LIN {X 0,Y 183.418,Z 1201.036,A -85,B 0,C 180,E1 27269.998,E2 27269.998} C_VEL
LIN {X 0,Y 183.226,Z 1199.826,A -85,B 0,C 180,E1 27279.492,E2 27279.492} C_VEL
LIN {X 0,Y 186.448,Z 1195.295,A -85,B 0,C 180,E1 27291.681,E2 27291.681} C_VEL
LIN {X 0,Y 197.947,Z 1184.674,A -85,B 0,C 180,E1 27306.27,E2 27306.27} C_VEL
LIN {X 0,Y 217.326,Z 1169.341,A -85,B 0,C 180,E1 27318.341,E2 27318.341} C_VEL
LIN {X 0,Y 246.49,Z 1146.185,A -85,B 0,C 180,E1 27329.12,E2 27329.12} C_VEL
LIN {X 0,Y 277.502,Z 1119.353,A -85,B 0,C 180,E1 27336.61,E2 27336.61} C_VEL
LIN {X 0,Y 311.114,Z 1086.295,A -85,B 0,C 180,E1 27342.398,E2 27342.398} C_VEL
LIN {X 0,Y 342.028,Z 1050.422,A -85,B 0,C 180,E1 27346.399,E2 27346.399} C_VEL
LIN {X 0,Y 359.417,Z 1027.318,A -85,B 0,C 180,E1 27348.285,E2 27348.285} C_VEL
LIN {X 0,Y 360.437,Z 1023.489,A -85,B 0,C 180,E1 27349.768,E2 27349.768} C_VEL
LIN {X 0,Y 361.093,Z 1015.57,A -85,B 0,C 180,E1 27355.186,E2 27355.186} C_VEL
LIN {X 0,Y 361.858,Z 1011.871,A -85,B 0,C 180,E1 27359.986,E2 27359.986} C_VEL
LIN {X 0,Y 359.734,Z 1016.107,A -85,B 0,C 180,E1 27365.978,E2 27365.978} C_VEL
LIN {X 0,Y 357.801,Z 1024.145,A -85,B 0,C 180,E1 27371.424,E2 27371.424} C_VEL
LIN {X 0,Y 356.491,Z 1027.72,A -85,B 0,C 180,E1 27372.861,E2 27372.861} C_VEL
LIN {X 0,Y 326.897,Z 1064.503,A -85,B 0,C 180,E1 27376.431,E2 27376.431} C_VEL
LIN {X 0,Y 295.294,Z 1097.247,A -85,B 0,C 180,E1 27381.232,E2 27381.232} C_VEL
LIN {X 0,Y 262.763,Z 1126.328,A -85,B 0,C 180,E1 27387.865,E2 27387.865} C_VEL
LIN {X 0,Y 231.737,Z 1150.541,A -85,B 0,C 180,E1 27397.047,E2 27397.047} C_VEL
LIN {X 0,Y 223.281,Z 1156.799,A -85,B 0,C 180,E1 27400.412,E2 27400.412} C_VEL
LIN {X 0,Y 211.981,Z 1163.134,A -85,B 0,C 180,E1 27403.536,E2 27403.536} C_VEL
LIN {X 0,Y 201.181,Z 1168.751,A -85,B 0,C 180,E1 27407.047,E2 27407.047} C_VEL
LIN {X 0,Y 184.669,Z 1180.419,A -85,B 0,C 180,E1 27420.598,E2 27420.598} C_VEL
LIN {X 0,Y 176.715,Z 1187.063,A -85,B 0,C 180,E1 27435.138,E2 27435.138} C_VEL
LIN {X 0,Y 175.238,Z 1188.956,A -85,B 0,C 180,E1 27445.056,E2 27445.056} C_VEL
LIN {X 0,Y 175.45,Z 1189.257,A -85,B 0,C 180,E1 27450.002,E2 27450.002} C_VEL
LIN {X 0,Y 175.659,Z 1188.194,A -85,B 0,C 180,E1 27459.91,E2 27459.91} C_VEL
LIN {X 0,Y 179.978,Z 1184.048,A -85,B 0,C 180,E1 27472.636,E2 27472.636} C_VEL
LIN {X 0,Y 191.782,Z 1175.244,A -85,B 0,C 180,E1 27486.227,E2 27486.227} C_VEL
LIN {X 0,Y 211.897,Z 1161.357,A -85,B 0,C 180,E1 27498.489,E2 27498.489} C_VEL
LIN {X 0,Y 239.263,Z 1141.674,A -85,B 0,C 180,E1 27508.501,E2 27508.501} C_VEL
LIN {X 0,Y 271.981,Z 1115.727,A -85,B 0,C 180,E1 27516.456,E2 27516.456} C_VEL
LIN {X 0,Y 305.801,Z 1084.371,A -85,B 0,C 180,E1 27522.269,E2 27522.269} C_VEL
LIN {X 0,Y 337.194,Z 1050.092,A -85,B 0,C 180,E1 27526.393,E2 27526.393} C_VEL
LIN {X 0,Y 351.788,Z 1031.697,A -85,B 0,C 180,E1 27528.002,E2 27528.002} C_VEL
LIN {X 0,Y 353.629,Z 1025.8,A -85,B 0,C 180,E1 27531.206,E2 27531.206} C_VEL
LIN {X 0,Y 355.183,Z 1021.103,A -85,B 0,C 180,E1 27535.134,E2 27535.134} C_VEL
LIN {X 0,Y 356.99,Z 1017.989,A -85,B 0,C 180,E1 27540.014,E2 27540.014} C_VEL
LIN {X 0,Y 356.017,Z 1023.243,A -85,B 0,C 180,E1 27546.105,E2 27546.105} C_VEL
LIN {X 0,Y 355.109,Z 1030.41,A -85,B 0,C 180,E1 27550.677,E2 27550.677} C_VEL
LIN {X 0,Y 325.133,Z 1067.904,A -85,B 0,C 180,E1 27554.017,E2 27554.017} C_VEL
LIN {X 0,Y 292.851,Z 1101.689,A -85,B 0,C 180,E1 27558.503,E2 27558.503} C_VEL
LIN {X 0,Y 258.573,Z 1132.56,A -85,B 0,C 180,E1 27565.062,E2 27565.062} C_VEL
LIN {X 0,Y 228.636,Z 1156.349,A -85,B 0,C 180,E1 27573.342,E2 27573.342} C_VEL
LIN {X 0,Y 201.93,Z 1176.328,A -85,B 0,C 180,E1 27585.022,E2 27585.022} C_VEL
LIN {X 0,Y 184.29,Z 1189.982,A -85,B 0,C 180,E1 27599.056,E2 27599.056} C_VEL
LIN {X 0,Y 177.725,Z 1196.4,A -85,B 0,C 180,E1 27610.114,E2 27610.114} C_VEL
LIN {X 0,Y 175.342,Z 1199.552,A -85,B 0,C 180,E1 27620.072,E2 27620.072} C_VEL
LIN {X 0,Y 175.506,Z 1200.777,A -85,B 0,C 180,E1 27629.998,E2 27629.998} C_VEL
LIN {X 0,Y 175.34,Z 1199.564,A -85,B 0,C 180,E1 27639.923,E2 27639.923} C_VEL
LIN {X 0,Y 178.183,Z 1195.845,A -85,B 0,C 180,E1 27651.053,E2 27651.053} C_VEL
LIN {X 0,Y 189.458,Z 1185.834,A -85,B 0,C 180,E1 27666.125,E2 27666.125} C_VEL
LIN {X 0,Y 210.379,Z 1170.234,A -85,B 0,C 180,E1 27679.33,E2 27679.33} C_VEL
LIN {X 0,Y 240.858,Z 1147.022,A -85,B 0,C 180,E1 27690.408,E2 27690.408} C_VEL
LIN {X 0,Y 271.953,Z 1121.223,A -85,B 0,C 180,E1 27697.745,E2 27697.745} C_VEL
LIN {X 0,Y 307.104,Z 1087.646,A -85,B 0,C 180,E1 27703.633,E2 27703.633} C_VEL
LIN {X 0,Y 339.058,Z 1051.582,A -85,B 0,C 180,E1 27707.614,E2 27707.614} C_VEL
LIN {X 0,Y 355.138,Z 1030.656,A -85,B 0,C 180,E1 27709.326,E2 27709.326} C_VEL
LIN {X 0,Y 356.13,Z 1023.435,A -85,B 0,C 180,E1 27713.897,E2 27713.897} C_VEL
LIN {X 0,Y 357.106,Z 1018.216,A -85,B 0,C 180,E1 27719.986,E2 27719.986} C_VEL
LIN {X 0,Y 354.832,Z 1022.647,A -85,B 0,C 180,E1 27726.097,E2 27726.097} C_VEL
LIN {X 0,Y 352.474,Z 1030.744,A -85,B 0,C 180,E1 27731.588,E2 27731.588} C_VEL
LIN {X 0,Y 349.194,Z 1035.472,A -85,B 0,C 180,E1 27732.186,E2 27732.186} C_VEL
LIN {X 0,Y 318.089,Z 1071.841,A -85,B 0,C 180,E1 27735.916,E2 27735.916} C_VEL
LIN {X 0,Y 285.251,Z 1104.275,A -85,B 0,C 180,E1 27740.988,E2 27740.988} C_VEL
LIN {X 0,Y 252.697,Z 1131.538,A -85,B 0,C 180,E1 27747.813,E2 27747.813} C_VEL
LIN {X 0,Y 223.071,Z 1153.62,A -85,B 0,C 180,E1 27756.775,E2 27756.775} C_VEL
LIN {X 0,Y 201.181,Z 1168.751,A -85,B 0,C 180,E1 27767.047,E2 27767.047} C_VEL
LIN {X 0,Y 190.976,Z 1173.788,A -85,B 0,C 180,E1 27770.964,E2 27770.964} C_VEL
LIN {X 0,Y 181.496,Z 1178.028,A -85,B 0,C 180,E1 27775.315,E2 27775.315} C_VEL
LIN {X 0,Y 170.975,Z 1185.702,A -85,B 0,C 180,E1 27789.299,E2 27789.299} C_VEL
LIN {X 0,Y 167.334,Z 1189.216,A -85,B 0,C 180,E1 27804.821,E2 27804.821} C_VEL
LIN {X 0,Y 167.543,Z 1189.516,A -85,B 0,C 180,E1 27810.003,E2 27810.003} C_VEL
LIN {X 0,Y 167.837,Z 1188.455,A -85,B 0,C 180,E1 27820.376,E2 27820.376} C_VEL
LIN {X 0,Y 173.857,Z 1183.357,A -85,B 0,C 180,E1 27835.762,E2 27835.762} C_VEL
LIN {X 0,Y 188.248,Z 1173.634,A -85,B 0,C 180,E1 27849.957,E2 27849.957} C_VEL
LIN {X 0,Y 212.732,Z 1157.426,A -85,B 0,C 180,E1 27862.766,E2 27862.766} C_VEL
LIN {X 0,Y 243.562,Z 1135.829,A -85,B 0,C 180,E1 27872.461,E2 27872.461} C_VEL
LIN {X 0,Y 277.925,Z 1108.195,A -85,B 0,C 180,E1 27879.707,E2 27879.707} C_VEL
LIN {X 0,Y 309.381,Z 1078.804,A -85,B 0,C 180,E1 27884.549,E2 27884.549} C_VEL
LIN {X 0,Y 341.478,Z 1042.944,A -85,B 0,C 180,E1 27888.385,E2 27888.385} C_VEL
LIN {X 0,Y 347.471,Z 1035.414,A -85,B 0,C 180,E1 27889.151,E2 27889.151} C_VEL
LIN {X 0,Y 350.105,Z 1027.407,A -85,B 0,C 180,E1 27895.063,E2 27895.063} C_VEL
LIN {X 0,Y 352.178,Z 1024.309,A -85,B 0,C 180,E1 27900.014,E2 27900.014} C_VEL
LIN {X 0,Y 350.951,Z 1029.552,A -85,B 0,C 180,E1 27906.193,E2 27906.193} C_VEL
LIN {X 0,Y 350.216,Z 1034.617,A -85,B 0,C 180,E1 27909.607,E2 27909.607} C_VEL
LIN {X 0,Y 319.882,Z 1071.453,A -85,B 0,C 180,E1 27913.008,E2 27913.008} C_VEL
LIN {X 0,Y 285.546,Z 1105.885,A -85,B 0,C 180,E1 27917.714,E2 27917.714} C_VEL
LIN {X 0,Y 252.287,Z 1134.637,A -85,B 0,C 180,E1 27924.013,E2 27924.013} C_VEL
LIN {X 0,Y 220.335,Z 1158.844,A -85,B 0,C 180,E1 27932.842,E2 27932.842} C_VEL
LIN {X 0,Y 193.955,Z 1177.619,A -85,B 0,C 180,E1 27944.552,E2 27944.552} C_VEL
LIN {X 0,Y 176.012,Z 1190.711,A -85,B 0,C 180,E1 27959.195,E2 27959.195} C_VEL
LIN {X 0,Y 170.118,Z 1196.133,A -85,B 0,C 180,E1 27969.185,E2 27969.185} C_VEL
LIN {X 0,Y 167.202,Z 1200.084,A -85,B 0,C 180,E1 27984.009,E2 27984.009} C_VEL
LIN {X 0,Y 167.594,Z 1200.517,A -85,B 0,C 180,E1 27989.997,E2 27989.997} C_VEL
LIN {X 0,Y 167.484,Z 1199.302,A -85,B 0,C 180,E1 28000.393,E2 28000.393} C_VEL
LIN {X 0,Y 171.231,Z 1194.909,A -85,B 0,C 180,E1 28013.396,E2 28013.396} C_VEL
LIN {X 0,Y 184.708,Z 1184.247,A -85,B 0,C 180,E1 28029.173,E2 28029.173} C_VEL
LIN {X 0,Y 206.114,Z 1169.15,A -85,B 0,C 180,E1 28041.594,E2 28041.594} C_VEL
LIN {X 0,Y 238.305,Z 1145.637,A -85,B 0,C 180,E1 28052.588,E2 28052.588} C_VEL
LIN {X 0,Y 271.532,Z 1118.598,A -85,B 0,C 180,E1 28059.899,E2 28059.899} C_VEL
LIN {X 0,Y 306.256,Z 1086.014,A -85,B 0,C 180,E1 28065.312,E2 28065.312} C_VEL
LIN {X 0,Y 338.54,Z 1049.89,A -85,B 0,C 180,E1 28069.104,E2 28069.104} C_VEL
LIN {X 0,Y 350.233,Z 1034.886,A -85,B 0,C 180,E1 28070.393,E2 28070.393} C_VEL
LIN {X 0,Y 351.273,Z 1028.329,A -85,B 0,C 180,E1 28075.051,E2 28075.051} C_VEL
LIN {X 0,Y 352.285,Z 1024.526,A -85,B 0,C 180,E1 28079.986,E2 28079.986} C_VEL
LIN {X 0,Y 349.637,Z 1029.052,A -85,B 0,C 180,E1 28086.266,E2 28086.266} C_VEL
LIN {X 0,Y 347.681,Z 1035.385,A -85,B 0,C 180,E1 28090.695,E2 28090.695} C_VEL
LIN {X 0,Y 339.539,Z 1045.579,A -85,B 0,C 180,E1 28091.739,E2 28091.739} C_VEL
LIN {X 0,Y 308.214,Z 1080.186,A -85,B 0,C 180,E1 28095.511,E2 28095.511} C_VEL
LIN {X 0,Y 273.406,Z 1112.194,A -85,B 0,C 180,E1 28101.002,E2 28101.002} C_VEL
LIN {X 0,Y 240.246,Z 1138.343,A -85,B 0,C 180,E1 28108.292,E2 28108.292} C_VEL
LIN {X 0,Y 208.56,Z 1160.321,A -85,B 0,C 180,E1 28118.845,E2 28118.845} C_VEL
LIN {X 0,Y 185.105,Z 1175.622,A -85,B 0,C 180,E1 28132.249,E2 28132.249} C_VEL
LIN {X 0,Y 181.496,Z 1178.028,A -85,B 0,C 180,E1 28135.315,E2 28135.315} C_VEL
LIN {X 0,Y 172.831,Z 1181.712,A -85,B 0,C 180,E1 28140.101,E2 28140.101} C_VEL
LIN {X 0,Y 165.053,Z 1184.714,A -85,B 0,C 180,E1 28145.359,E2 28145.359} C_VEL
LIN {X 0,Y 159.959,Z 1188.748,A -85,B 0,C 180,E1 28159.112,E2 28159.112} C_VEL
LIN {X 0,Y 159.653,Z 1189.775,A -85,B 0,C 180,E1 28170.003,E2 28170.003} C_VEL
LIN {X 0,Y 159.995,Z 1188.718,A -85,B 0,C 180,E1 28180.891,E2 28180.891} C_VEL
LIN {X 0,Y 166.618,Z 1183.622,A -85,B 0,C 180,E1 28196.969,E2 28196.969} C_VEL
LIN {X 0,Y 182.326,Z 1173.712,A -85,B 0,C 180,E1 28211.811,E2 28211.811} C_VEL
LIN {X 0,Y 208.771,Z 1157.113,A -85,B 0,C 180,E1 28224.926,E2 28224.926} C_VEL
LIN {X 0,Y 239.408,Z 1136.456,A -85,B 0,C 180,E1 28234.085,E2 28234.085} C_VEL
LIN {X 0,Y 275.19,Z 1108.466,A -85,B 0,C 180,E1 28241.308,E2 28241.308} C_VEL
LIN {X 0,Y 307.049,Z 1079.349,A -85,B 0,C 180,E1 28245.977,E2 28245.977} C_VEL
LIN {X 0,Y 339.271,Z 1044.02,A -85,B 0,C 180,E1 28249.649,E2 28249.649} C_VEL
LIN {X 0,Y 342.654,Z 1039.794,A -85,B 0,C 180,E1 28250.177,E2 28250.177} C_VEL
LIN {X 0,Y 344.976,Z 1033.672,A -85,B 0,C 180,E1 28254.989,E2 28254.989} C_VEL
LIN {X 0,Y 347.141,Z 1030.439,A -85,B 0,C 180,E1 28260.014,E2 28260.014} C_VEL
LIN {X 0,Y 345.802,Z 1035.856,A -85,B 0,C 180,E1 28266.286,E2 28266.286} C_VEL
LIN {X 0,Y 345.346,Z 1038.832,A -85,B 0,C 180,E1 28268.419,E2 28268.419} C_VEL
LIN {X 0,Y 342.797,Z 1042.436,A -85,B 0,C 180,E1 28268.971,E2 28268.971} C_VEL
LIN {X 0,Y 309.616,Z 1080.038,A -85,B 0,C 180,E1 28272.54,E2 28272.54} C_VEL
LIN {X 0,Y 276.824,Z 1111.353,A -85,B 0,C 180,E1 28277.114,E2 28277.114} C_VEL
LIN {X 0,Y 240.003,Z 1141.226,A -85,B 0,C 180,E1 28284.302,E2 28284.302} C_VEL
LIN {X 0,Y 208.261,Z 1163.884,A -85,B 0,C 180,E1 28293.675,E2 28293.675} C_VEL
LIN {X 0,Y 181.804,Z 1181.601,A -85,B 0,C 180,E1 28306.704,E2 28306.704} C_VEL
LIN {X 0,Y 166.925,Z 1192.112,A -85,B 0,C 180,E1 28320.422,E2 28320.422} C_VEL
LIN {X 0,Y 160.615,Z 1197.691,A -85,B 0,C 180,E1 28333.603,E2 28333.603} C_VEL
LIN {X 0,Y 159.344,Z 1199.885,A -85,B 0,C 180,E1 28344.556,E2 28344.556} C_VEL
LIN {X 0,Y 159.704,Z 1200.258,A -85,B 0,C 180,E1 28349.997,E2 28349.997} C_VEL
LIN {X 0,Y 159.61,Z 1199.039,A -85,B 0,C 180,E1 28360.912,E2 28360.912} C_VEL
LIN {X 0,Y 163.791,Z 1194.642,A -85,B 0,C 180,E1 28374.527,E2 28374.527} C_VEL
LIN {X 0,Y 178.314,Z 1184.017,A -85,B 0,C 180,E1 28390.801,E2 28390.801} C_VEL
LIN {X 0,Y 201.123,Z 1168.817,A -85,B 0,C 180,E1 28403.493,E2 28403.493} C_VEL
LIN {X 0,Y 234.583,Z 1145.365,A -85,B 0,C 180,E1 28414.396,E2 28414.396} C_VEL
LIN {X 0,Y 268.796,Z 1118.328,A -85,B 0,C 180,E1 28421.558,E2 28421.558} C_VEL
LIN {X 0,Y 305.061,Z 1084.991,A -85,B 0,C 180,E1 28426.906,E2 28426.906} C_VEL
LIN {X 0,Y 338.823,Z 1047.512,A -85,B 0,C 180,E1 28430.647,E2 28430.647} C_VEL
LIN {X 0,Y 345.344,Z 1039.407,A -85,B 0,C 180,E1 28431.366,E2 28431.366} C_VEL
LIN {X 0,Y 346.403,Z 1033.254,A -85,B 0,C 180,E1 28436.34,E2 28436.34} C_VEL
LIN {X 0,Y 347.248,Z 1030.655,A -85,B 0,C 180,E1 28439.986,E2 28439.986} C_VEL
LIN {X 0,Y 344.48,Z 1035.364,A -85,B 0,C 180,E1 28446.36,E2 28446.36} C_VEL
LIN {X 0,Y 342.916,Z 1039.568,A -85,B 0,C 180,E1 28449.496,E2 28449.496} C_VEL
LIN {X 0,Y 341.986,Z 1041.044,A -85,B 0,C 180,E1 28449.984,E2 28449.984} C_VEL
LIN {X 0,Y 308.561,Z 1077.993,A -85,B 0,C 180,E1 28453.732,E2 28453.732} C_VEL
LIN {X 0,Y 275.072,Z 1108.73,A -85,B 0,C 180,E1 28458.63,E2 28458.63} C_VEL
LIN {X 0,Y 239.268,Z 1136.669,A -85,B 0,C 180,E1 28465.851,E2 28465.851} C_VEL
LIN {X 0,Y 206.737,Z 1158.483,A -85,B 0,C 180,E1 28475.75,E2 28475.75} C_VEL
LIN {X 0,Y 181.917,Z 1174.027,A -85,B 0,C 180,E1 28488.357,E2 28488.357} C_VEL
LIN {X 0,Y 166.587,Z 1183.689,A -85,B 0,C 180,E1 28503.031,E2 28503.031} C_VEL
LIN {X 0,Y 165.053,Z 1184.714,A -85,B 0,C 180,E1 28505.359,E2 28505.359} C_VEL
LIN {X 0,Y 160.242,Z 1186.573,A -85,B 0,C 180,E1 28509.619,E2 28509.619} C_VEL
LIN {X 0,Y 152.607,Z 1188.636,A -85,B 0,C 180,E1 28516.32,E2 28516.32} C_VEL
LIN {X 0,Y 152.35,Z 1188.726,A -85,B 0,C 180,E1 28517.141,E2 28517.141} C_VEL
LIN {X 0,Y 151.743,Z 1190.035,A -85,B 0,C 180,E1 28530.003,E2 28530.003} C_VEL
LIN {X 0,Y 152.168,Z 1188.98,A -85,B 0,C 180,E1 28541.459,E2 28541.459} C_VEL
LIN {X 0,Y 156.867,Z 1185.546,A -85,B 0,C 180,E1 28554.346,E2 28554.346} C_VEL
LIN {X 0,Y 172.503,Z 1176.107,A -85,B 0,C 180,E1 28570.973,E2 28570.973} C_VEL
LIN {X 0,Y 196.444,Z 1162.169,A -85,B 0,C 180,E1 28583.875,E2 28583.875} C_VEL
LIN {X 0,Y 230.049,Z 1140.657,A -85,B 0,C 180,E1 28594.508,E2 28594.508} C_VEL
LIN {X 0,Y 263.658,Z 1116.101,A -85,B 0,C 180,E1 28601.467,E2 28601.467} C_VEL
LIN {X 0,Y 299.879,Z 1084.608,A -85,B 0,C 180,E1 28606.805,E2 28606.805} C_VEL
LIN {X 0,Y 332.328,Z 1050.899,A -85,B 0,C 180,E1 28610.458,E2 28610.458} C_VEL
LIN {X 0,Y 336.705,Z 1045.714,A -85,B 0,C 180,E1 28610.884,E2 28610.884} C_VEL
LIN {X 0,Y 338.021,Z 1043.677,A -85,B 0,C 180,E1 28611.615,E2 28611.615} C_VEL
LIN {X 0,Y 340.938,Z 1037.886,A -85,B 0,C 180,E1 28617.475,E2 28617.475} C_VEL
LIN {X 0,Y 342.105,Z 1036.566,A -85,B 0,C 180,E1 28620.015,E2 28620.015} C_VEL
LIN {X 0,Y 340.561,Z 1042.087,A -85,B 0,C 180,E1 28626.383,E2 28626.383} C_VEL
LIN {X 0,Y 340.181,Z 1043.798,A -85,B 0,C 180,E1 28627.672,E2 28627.672} C_VEL
LIN {X 0,Y 305.455,Z 1082.322,A -85,B 0,C 180,E1 28631.328,E2 28631.328} C_VEL
LIN {X 0,Y 271.242,Z 1113.777,A -85,B 0,C 180,E1 28635.963,E2 28635.963} C_VEL
LIN {X 0,Y 236.17,Z 1141.359,A -85,B 0,C 180,E1 28642.596,E2 28642.596} C_VEL
LIN {X 0,Y 204.395,Z 1163.218,A -85,B 0,C 180,E1 28651.512,E2 28651.512} C_VEL
LIN {X 0,Y 175.581,Z 1181.505,A -85,B 0,C 180,E1 28665.023,E2 28665.023} C_VEL
LIN {X 0,Y 158.08,Z 1193.072,A -85,B 0,C 180,E1 28681.445,E2 28681.445} C_VEL
LIN {X 0,Y 152.905,Z 1197.427,A -85,B 0,C 180,E1 28692.751,E2 28692.751} C_VEL
LIN {X 0,Y 151.441,Z 1199.782,A -85,B 0,C 180,E1 28706.634,E2 28706.634} C_VEL
LIN {X 0,Y 151.448,Z 1199.783,A -85,B 0,C 180,E1 28713.413,E2 28713.413} C_VEL
LIN {X 0,Y 152.901,Z 1197.448,A -85,B 0,C 180,E1 28727.244,E2 28727.244} C_VEL
LIN {X 0,Y 162.327,Z 1190.096,A -85,B 0,C 180,E1 28743.952,E2 28743.952} C_VEL
LIN {X 0,Y 183.516,Z 1176.639,A -85,B 0,C 180,E1 28759.608,E2 28759.608} C_VEL
LIN {X 0,Y 214.42,Z 1156.611,A -85,B 0,C 180,E1 28771.751,E2 28771.751} C_VEL
LIN {X 0,Y 249.177,Z 1131.765,A -85,B 0,C 180,E1 28780.16,E2 28780.16} C_VEL
LIN {X 0,Y 286.715,Z 1100.365,A -85,B 0,C 180,E1 28786.319,E2 28786.319} C_VEL
LIN {X 0,Y 320.047,Z 1067.342,A -85,B 0,C 180,E1 28790.263,E2 28790.263} C_VEL
LIN {X 0,Y 340.258,Z 1043.985,A -85,B 0,C 180,E1 28792.33,E2 28792.33} C_VEL
LIN {X 0,Y 341.548,Z 1038.489,A -85,B 0,C 180,E1 28797.45,E2 28797.45} C_VEL
LIN {X 0,Y 342.211,Z 1036.783,A -85,B 0,C 180,E1 28799.985,E2 28799.985} C_VEL
LIN {X 0,Y 339.167,Z 1041.456,A -85,B 0,C 180,E1 28806.379,E2 28806.379} C_VEL
LIN {X 0,Y 337.889,Z 1044.452,A -85,B 0,C 180,E1 28808.734,E2 28808.734} C_VEL
LIN {X 0,Y 326.122,Z 1058.025,A -85,B 0,C 180,E1 28810.102,E2 28810.102} C_VEL
LIN {X 0,Y 292.161,Z 1092.097,A -85,B 0,C 180,E1 28814.127,E2 28814.127} C_VEL
LIN {X 0,Y 256.786,Z 1121.504,A -85,B 0,C 180,E1 28819.691,E2 28819.691} C_VEL
LIN {X 0,Y 221.694,Z 1146.471,A -85,B 0,C 180,E1 28827.616,E2 28827.616} C_VEL
LIN {X 0,Y 191.794,Z 1164.903,A -85,B 0,C 180,E1 28838.016,E2 28838.016} C_VEL
LIN {X 0,Y 169.317,Z 1178.006,A -85,B 0,C 180,E1 28851.341,E2 28851.341} C_VEL
LIN {X 0,Y 156.027,Z 1186.229,A -85,B 0,C 180,E1 28867.21,E2 28867.21} C_VEL
LIN {X 0,Y 152.35,Z 1188.726,A -85,B 0,C 180,E1 28877.141,E2 28877.141} C_VEL
LIN {X 0,Y 149.463,Z 1189.68,A -85,B 0,C 180,E1 28881.973,E2 28881.973} C_VEL
LIN {X 0,Y 143.783,Z 1190.277,A -85,B 0,C 180,E1 28890.351,E2 28890.351} C_VEL
LIN {X 0,Y 144.349,Z 1189.242,A -85,B 0,C 180,E1 28902.088,E2 28902.088} C_VEL
LIN {X 0,Y 150.329,Z 1185.303,A -85,B 0,C 180,E1 28916.897,E2 28916.897} C_VEL
LIN {X 0,Y 168.326,Z 1175.37,A -85,B 0,C 180,E1 28934.146,E2 28934.146} C_VEL
LIN {X 0,Y 195.503,Z 1160.167,A -85,B 0,C 180,E1 28947.28,E2 28947.28} C_VEL
LIN {X 0,Y 229.718,Z 1138.958,A -85,B 0,C 180,E1 28957.068,E2 28957.068} C_VEL
LIN {X 0,Y 265.483,Z 1112.928,A -85,B 0,C 180,E1 28963.829,E2 28963.829} C_VEL
LIN {X 0,Y 302.055,Z 1081.275,A -85,B 0,C 180,E1 28968.785,E2 28968.785} C_VEL
LIN {X 0,Y 331.696,Z 1050.45,A -85,B 0,C 180,E1 28971.894,E2 28971.894} C_VEL
LIN {X 0,Y 332.878,Z 1048.939,A -85,B 0,C 180,E1 28972.189,E2 28972.189} C_VEL
LIN {X 0,Y 335.59,Z 1043.877,A -85,B 0,C 180,E1 28977.434,E2 28977.434} C_VEL
LIN {X 0,Y 336.892,Z 1042.561,A -85,B 0,C 180,E1 28980.015,E2 28980.015} C_VEL
LIN {X 0,Y 335.279,Z 1047.524,A -85,B 0,C 180,E1 28985.966,E2 28985.966} C_VEL
LIN {X 0,Y 334.778,Z 1048.798,A -85,B 0,C 180,E1 28986.758,E2 28986.758} C_VEL
LIN {X 0,Y 301.437,Z 1084.552,A -85,B 0,C 180,E1 28990.081,E2 28990.081} C_VEL
LIN {X 0,Y 265.694,Z 1116.276,A -85,B 0,C 180,E1 28994.786,E2 28994.786} C_VEL
LIN {X 0,Y 230.499,Z 1142.98,A -85,B 0,C 180,E1 29001.267,E2 29001.267} C_VEL
LIN {X 0,Y 196.334,Z 1165.26,A -85,B 0,C 180,E1 29010.774,E2 29010.774} C_VEL
LIN {X 0,Y 168.213,Z 1182.24,A -85,B 0,C 180,E1 29024.052,E2 29024.052} C_VEL
LIN {X 0,Y 150.951,Z 1192.803,A -85,B 0,C 180,E1 29039.962,E2 29039.962} C_VEL
LIN {X 0,Y 145.206,Z 1197.161,A -85,B 0,C 180,E1 29051.805,E2 29051.805} C_VEL
LIN {X 0,Y 143.513,Z 1199.363,A -85,B 0,C 180,E1 29063.953,E2 29063.953} C_VEL
LIN {X 0,Y 143.88,Z 1199.739,A -85,B 0,C 180,E1 29069.997,E2 29069.997} C_VEL
LIN {X 0,Y 143.9,Z 1198.514,A -85,B 0,C 180,E1 29082.121,E2 29082.121} C_VEL
LIN {X 0,Y 149.11,Z 1194.108,A -85,B 0,C 180,E1 29097.129,E2 29097.129} C_VEL
LIN {X 0,Y 165.07,Z 1184.082,A -85,B 0,C 180,E1 29113.789,E2 29113.789} C_VEL
LIN {X 0,Y 190.247,Z 1169.19,A -85,B 0,C 180,E1 29126.943,E2 29126.943} C_VEL
LIN {X 0,Y 224.909,Z 1146.812,A -85,B 0,C 180,E1 29137.488,E2 29137.488} C_VEL
LIN {X 0,Y 260.749,Z 1120.48,A -85,B 0,C 180,E1 29144.458,E2 29144.458} C_VEL
LIN {X 0,Y 298.136,Z 1087.828,A -85,B 0,C 180,E1 29149.554,E2 29149.554} C_VEL
LIN {X 0,Y 331.191,Z 1053.334,A -85,B 0,C 180,E1 29152.91,E2 29152.91} C_VEL
LIN {X 0,Y 334.77,Z 1049.095,A -85,B 0,C 180,E1 29153.231,E2 29153.231} C_VEL
LIN {X 0,Y 336.235,Z 1044.474,A -85,B 0,C 180,E1 29157.41,E2 29157.41} C_VEL
LIN {X 0,Y 336.979,Z 1042.777,A -85,B 0,C 180,E1 29159.985,E2 29159.985} C_VEL
LIN {X 0,Y 333.697,Z 1047.565,A -85,B 0,C 180,E1 29166.483,E2 29166.483} C_VEL
LIN {X 0,Y 332.952,Z 1049.206,A -85,B 0,C 180,E1 29167.809,E2 29167.809} C_VEL
LIN {X 0,Y 299.915,Z 1083.443,A -85,B 0,C 180,E1 29171.366,E2 29171.366} C_VEL
LIN {X 0,Y 262.037,Z 1115.853,A -85,B 0,C 180,E1 29176.62,E2 29176.62} C_VEL
LIN {X 0,Y 226.514,Z 1141.125,A -85,B 0,C 180,E1 29183.568,E2 29183.568} C_VEL
LIN {X 0,Y 192.871,Z 1161.83,A -85,B 0,C 180,E1 29193.596,E2 29193.596} C_VEL
LIN {X 0,Y 165.449,Z 1176.928,A -85,B 0,C 180,E1 29207.739,E2 29207.739} C_VEL
LIN {X 0,Y 150.301,Z 1185.369,A -85,B 0,C 180,E1 29223.104,E2 29223.104} C_VEL
LIN {X 0,Y 144.318,Z 1189.271,A -85,B 0,C 180,E1 29237.915,E2 29237.915} C_VEL
LIN {X 0,Y 143.783,Z 1190.277,A -85,B 0,C 180,E1 29250.351,E2 29250.351} C_VEL
LIN {X 0,Y 141.037,Z 1190.14,A -85,B 0,C 180,E1 29255.503,E2 29255.503} C_VEL
LIN {X 0,Y 136.867,Z 1189.203,A -85,B 0,C 180,E1 29264.429,E2 29264.429} C_VEL
LIN {X 0,Y 145.349,Z 1184.423,A -85,B 0,C 180,E1 29281.324,E2 29281.324} C_VEL
LIN {X 0,Y 164.419,Z 1174.716,A -85,B 0,C 180,E1 29297.332,E2 29297.332} C_VEL
LIN {X 0,Y 195.011,Z 1158.263,A -85,B 0,C 180,E1 29310.667,E2 29310.667} C_VEL
LIN {X 0,Y 229.691,Z 1137.268,A -85,B 0,C 180,E1 29319.64,E2 29319.64} C_VEL
LIN {X 0,Y 267.76,Z 1109.714,A -85,B 0,C 180,E1 29326.212,E2 29326.212} C_VEL
LIN {X 0,Y 302.466,Z 1079.762,A -85,B 0,C 180,E1 29330.516,E2 29330.516} C_VEL
LIN {X 0,Y 327.027,Z 1054.72,A -85,B 0,C 180,E1 29332.968,E2 29332.968} C_VEL
LIN {X 0,Y 328.228,Z 1053.18,A -85,B 0,C 180,E1 29333.635,E2 29333.635} C_VEL
LIN {X 0,Y 331.562,Z 1048.479,A -85,B 0,C 180,E1 29340.015,E2 29340.015} C_VEL
LIN {X 0,Y 329.994,Z 1053.034,A -85,B 0,C 180,E1 29345.598,E2 29345.598} C_VEL
LIN {X 0,Y 296.687,Z 1087.417,A -85,B 0,C 180,E1 29348.891,E2 29348.891} C_VEL
LIN {X 0,Y 258.54,Z 1120.147,A -85,B 0,C 180,E1 29353.797,E2 29353.797} C_VEL
LIN {X 0,Y 221.87,Z 1146.427,A -85,B 0,C 180,E1 29360.526,E2 29360.526} C_VEL
LIN {X 0,Y 187.852,Z 1167.584,A -85,B 0,C 180,E1 29370.142,E2 29370.142} C_VEL
LIN {X 0,Y 160.609,Z 1182.994,A -85,B 0,C 180,E1 29383.18,E2 29383.18} C_VEL
LIN {X 0,Y 141.894,Z 1193.807,A -85,B 0,C 180,E1 29401.361,E2 29401.361} C_VEL
LIN {X 0,Y 136.083,Z 1198.237,A -85,B 0,C 180,E1 29417.165,E2 29417.165} C_VEL
LIN {X 0,Y 135.979,Z 1199.479,A -85,B 0,C 180,E1 29429.997,E2 29429.997} C_VEL
LIN {X 0,Y 136.08,Z 1198.251,A -85,B 0,C 180,E1 29442.829,E2 29442.829} C_VEL
LIN {X 0,Y 141.896,Z 1193.841,A -85,B 0,C 180,E1 29458.631,E2 29458.631} C_VEL
LIN {X 0,Y 160.61,Z 1183.048,A -85,B 0,C 180,E1 29476.812,E2 29476.812} C_VEL
LIN {X 0,Y 187.872,Z 1167.677,A -85,B 0,C 180,E1 29489.839,E2 29489.839} C_VEL
LIN {X 0,Y 224.938,Z 1144.552,A -85,B 0,C 180,E1 29500.131,E2 29500.131} C_VEL
LIN {X 0,Y 261.3,Z 1118.089,A -85,B 0,C 180,E1 29506.607,E2 29506.607} C_VEL
LIN {X 0,Y 299.446,Z 1085.098,A -85,B 0,C 180,E1 29511.389,E2 29511.389} C_VEL
LIN {X 0,Y 330.055,Z 1053.25,A -85,B 0,C 180,E1 29514.403,E2 29514.403} C_VEL
LIN {X 0,Y 331.658,Z 1048.684,A -85,B 0,C 180,E1 29519.985,E2 29519.985} C_VEL
LIN {X 0,Y 328.253,Z 1053.515,A -85,B 0,C 180,E1 29526.467,E2 29526.467} C_VEL
LIN {X 0,Y 325.853,Z 1056.244,A -85,B 0,C 180,E1 29527.08,E2 29527.08} C_VEL
LIN {X 0,Y 290.324,Z 1091.055,A -85,B 0,C 180,E1 29530.765,E2 29530.765} C_VEL
LIN {X 0,Y 255.096,Z 1119.601,A -85,B 0,C 180,E1 29535.613,E2 29535.613} C_VEL
LIN {X 0,Y 216.487,Z 1145.761,A -85,B 0,C 180,E1 29543.225,E2 29543.225} C_VEL
LIN {X 0,Y 185.919,Z 1163.457,A -85,B 0,C 180,E1 29552.446,E2 29552.446} C_VEL
LIN {X 0,Y 156.879,Z 1178.541,A -85,B 0,C 180,E1 29567.607,E2 29567.607} C_VEL
LIN {X 0,Y 141.283,Z 1186.758,A -85,B 0,C 180,E1 29584.674,E2 29584.674} C_VEL
LIN {X 0,Y 135.766,Z 1190.257,A -85,B 0,C 180,E1 29603.613,E2 29603.613} C_VEL
LIN {X 0,Y 135.897,Z 1190.541,A -85,B 0,C 180,E1 29610.325,E2 29610.325} C_VEL
LIN {X 0,Y 136.867,Z 1189.203,A -85,B 0,C 180,E1 29624.429,E2 29624.429} C_VEL
LIN {X 0,Y 136.625,Z 1188.691,A -85,B 0,C 180,E1 29628.088,E2 29628.088} C_VEL
LIN {X 0,Y 135.029,Z 1186.446,A -85,B 0,C 180,E1 29638.296,E2 29638.296} C_VEL
LIN {X 0,Y 135.54,Z 1186.121,A -85,B 0,C 180,E1 29639.195,E2 29639.195} C_VEL
LIN {X 0,Y 154.68,Z 1176.957,A -85,B 0,C 180,E1 29656.906,E2 29656.906} C_VEL
LIN {X 0,Y 184.241,Z 1162.299,A -85,B 0,C 180,E1 29670.556,E2 29670.556} C_VEL
LIN {X 0,Y 222.121,Z 1140.531,A -85,B 0,C 180,E1 29680.605,E2 29680.605} C_VEL
LIN {X 0,Y 258.114,Z 1116,A -85,B 0,C 180,E1 29686.812,E2 29686.812} C_VEL
LIN {X 0,Y 296.06,Z 1084.708,A -85,B 0,C 180,E1 29691.507,E2 29691.507} C_VEL
LIN {X 0,Y 322.01,Z 1059.301,A -85,B 0,C 180,E1 29694.025,E2 29694.025} C_VEL
LIN {X 0,Y 323.18,Z 1057.881,A -85,B 0,C 180,E1 29694.65,E2 29694.65} C_VEL
LIN {X 0,Y 326.214,Z 1054.382,A -85,B 0,C 180,E1 29700.015,E2 29700.015} C_VEL
LIN {X 0,Y 324.751,Z 1057.797,A -85,B 0,C 180,E1 29704.614,E2 29704.614} C_VEL
LIN {X 0,Y 286.33,Z 1095.532,A -85,B 0,C 180,E1 29708.286,E2 29708.286} C_VEL
LIN {X 0,Y 248.372,Z 1126.018,A -85,B 0,C 180,E1 29713.225,E2 29713.225} C_VEL
LIN {X 0,Y 209.818,Z 1152.121,A -85,B 0,C 180,E1 29720.561,E2 29720.561} C_VEL
LIN {X 0,Y 174.396,Z 1172.422,A -85,B 0,C 180,E1 29731.354,E2 29731.354} C_VEL
LIN {X 0,Y 148.278,Z 1186.239,A -85,B 0,C 180,E1 29745.551,E2 29745.551} C_VEL
LIN {X 0,Y 132.881,Z 1194.796,A -85,B 0,C 180,E1 29762.939,E2 29762.939} C_VEL
LIN {X 0,Y 128.263,Z 1197.973,A -85,B 0,C 180,E1 29776.368,E2 29776.368} C_VEL
LIN {X 0,Y 128.059,Z 1199.219,A -85,B 0,C 180,E1 29789.997,E2 29789.997} C_VEL
LIN {X 0,Y 128.259,Z 1197.987,A -85,B 0,C 180,E1 29803.625,E2 29803.625} C_VEL
LIN {X 0,Y 134.773,Z 1193.573,A -85,B 0,C 180,E1 29820.298,E2 29820.298} C_VEL
LIN {X 0,Y 155.043,Z 1182.776,A -85,B 0,C 180,E1 29839.051,E2 29839.051} C_VEL
LIN {X 0,Y 183.83,Z 1167.406,A -85,B 0,C 180,E1 29852.083,E2 29852.083} C_VEL
LIN {X 0,Y 222.248,Z 1144.28,A -85,B 0,C 180,E1 29862.149,E2 29862.149} C_VEL
LIN {X 0,Y 259.516,Z 1117.821,A -85,B 0,C 180,E1 29868.377,E2 29868.377} C_VEL
LIN {X 0,Y 298.626,Z 1084.564,A -85,B 0,C 180,E1 29872.973,E2 29872.973} C_VEL
LIN {X 0,Y 324.802,Z 1058.01,A -85,B 0,C 180,E1 29875.383,E2 29875.383} C_VEL
LIN {X 0,Y 326.303,Z 1054.575,A -85,B 0,C 180,E1 29879.985,E2 29879.985} C_VEL
LIN {X 0,Y 323.066,Z 1058.428,A -85,B 0,C 180,E1 29885.688,E2 29885.688} C_VEL
LIN {X 0,Y 287.161,Z 1092.894,A -85,B 0,C 180,E1 29889.375,E2 29889.375} C_VEL
LIN {X 0,Y 249.563,Z 1122.307,A -85,B 0,C 180,E1 29894.356,E2 29894.356} C_VEL
LIN {X 0,Y 211.367,Z 1147.278,A -85,B 0,C 180,E1 29901.664,E2 29901.664} C_VEL
LIN {X 0,Y 175.115,Z 1167.004,A -85,B 0,C 180,E1 29912.722,E2 29912.722} C_VEL
LIN {X 0,Y 150.945,Z 1178.809,A -85,B 0,C 180,E1 29925.515,E2 29925.515} C_VEL
LIN {X 0,Y 134.015,Z 1187.023,A -85,B 0,C 180,E1 29943.194,E2 29943.194} C_VEL
LIN {X 0,Y 127.872,Z 1190.518,A -85,B 0,C 180,E1 29963.217,E2 29963.217} C_VEL
LIN {X 0,Y 128.057,Z 1190.812,A -85,B 0,C 180,E1 29970.003,E2 29970.003} C_VEL
LIN {X 0,Y 129.003,Z 1189.565,A -85,B 0,C 180,E1 29984.744,E2 29984.744} C_VEL
LIN {X 0,Y 135.54,Z 1186.121,A -85,B 0,C 180,E1 29999.195,E2 29999.195} C_VEL
LIN {X 0,Y 136.939,Z 1184.97,A -85,B 0,C 180,E1 30002.793,E2 30002.793} C_VEL
LIN {X 0,Y 139.942,Z 1181.382,A -85,B 0,C 180,E1 30012.672,E2 30012.672} C_VEL
LIN {X 0,Y 140.862,Z 1180.974,A -85,B 0,C 180,E1 30013.473,E2 30013.473} C_VEL
LIN {X 0,Y 168.284,Z 1168.433,A -85,B 0,C 180,E1 30028.551,E2 30028.551} C_VEL
LIN {X 0,Y 205.461,Z 1149.081,A -85,B 0,C 180,E1 30039.679,E2 30039.679} C_VEL
LIN {X 0,Y 242.669,Z 1125.886,A -85,B 0,C 180,E1 30046.657,E2 30046.657} C_VEL
LIN {X 0,Y 282.462,Z 1095.849,A -85,B 0,C 180,E1 30051.784,E2 30051.784} C_VEL
LIN {X 0,Y 317.865,Z 1063.077,A -85,B 0,C 180,E1 30055.244,E2 30055.244} C_VEL
LIN {X 0,Y 320.607,Z 1060.066,A -85,B 0,C 180,E1 30060.016,E2 30060.016} C_VEL
LIN {X 0,Y 319.552,Z 1062.296,A -85,B 0,C 180,E1 30063.33,E2 30063.33} C_VEL
LIN {X 0,Y 313.827,Z 1068.457,A -85,B 0,C 180,E1 30064.034,E2 30064.034} C_VEL
LIN {X 0,Y 276.311,Z 1102.759,A -85,B 0,C 180,E1 30067.581,E2 30067.581} C_VEL
LIN {X 0,Y 237.781,Z 1132.083,A -85,B 0,C 180,E1 30072.679,E2 30072.679} C_VEL
LIN {X 0,Y 198.674,Z 1156.65,A -85,B 0,C 180,E1 30080.348,E2 30080.348} C_VEL
LIN {X 0,Y 163.45,Z 1175.722,A -85,B 0,C 180,E1 30091.723,E2 30091.723} C_VEL
LIN {X 0,Y 136.211,Z 1188.97,A -85,B 0,C 180,E1 30108.265,E2 30108.265} C_VEL
LIN {X 0,Y 122.4,Z 1196.364,A -85,B 0,C 180,E1 30128.258,E2 30128.258} C_VEL
LIN {X 0,Y 119.792,Z 1198.579,A -85,B 0,C 180,E1 30142.749,E2 30142.749} C_VEL
LIN {X 0,Y 120.151,Z 1198.96,A -85,B 0,C 180,E1 30149.996,E2 30149.996} C_VEL
LIN {X 0,Y 120.463,Z 1197.724,A -85,B 0,C 180,E1 30164.526,E2 30164.526} C_VEL
LIN {X 0,Y 127.78,Z 1193.305,A -85,B 0,C 180,E1 30182.148,E2 30182.148} C_VEL
LIN {X 0,Y 149.726,Z 1182.504,A -85,B 0,C 180,E1 30201.455,E2 30201.455} C_VEL
LIN {X 0,Y 180.078,Z 1167.133,A -85,B 0,C 180,E1 30214.427,E2 30214.427} C_VEL
LIN {X 0,Y 219.847,Z 1144.01,A -85,B 0,C 180,E1 30224.206,E2 30224.206} C_VEL
LIN {X 0,Y 258.469,Z 1117.162,A -85,B 0,C 180,E1 30230.253,E2 30230.253} C_VEL
LIN {X 0,Y 297.212,Z 1084.762,A -85,B 0,C 180,E1 30234.495,E2 30234.495} C_VEL
LIN {X 0,Y 317.992,Z 1064.339,A -85,B 0,C 180,E1 30236.29,E2 30236.29} C_VEL
LIN {X 0,Y 319.605,Z 1062.513,A -85,B 0,C 180,E1 30236.666,E2 30236.666} C_VEL
LIN {X 0,Y 320.693,Z 1060.262,A -85,B 0,C 180,E1 30239.984,E2 30239.984} C_VEL
LIN {X 0,Y 317.973,Z 1063.27,A -85,B 0,C 180,E1 30244.754,E2 30244.754} C_VEL
LIN {X 0,Y 283.487,Z 1095.23,A -85,B 0,C 180,E1 30248.023,E2 30248.023} C_VEL
LIN {X 0,Y 244.276,Z 1124.928,A -85,B 0,C 180,E1 30253.024,E2 30253.024} C_VEL
LIN {X 0,Y 208.462,Z 1147.547,A -85,B 0,C 180,E1 30259.556,E2 30259.556} C_VEL
LIN {X 0,Y 170.805,Z 1167.273,A -85,B 0,C 180,E1 30270.397,E2 30270.397} C_VEL
LIN {X 0,Y 145.222,Z 1179.076,A -85,B 0,C 180,E1 30283.253,E2 30283.253} C_VEL
LIN {X 0,Y 126.845,Z 1187.289,A -85,B 0,C 180,E1 30301.545,E2 30301.545} C_VEL
LIN {X 0,Y 120,Z 1190.778,A -85,B 0,C 180,E1 30322.769,E2 30322.769} C_VEL
LIN {X 0,Y 120.162,Z 1191.071,A -85,B 0,C 180,E1 30330.004,E2 30330.004} C_VEL
LIN {X 0,Y 121.025,Z 1190.029,A -85,B 0,C 180,E1 30344.464,E2 30344.464} C_VEL
LIN {X 0,Y 131.752,Z 1184.956,A -85,B 0,C 180,E1 30364.996,E2 30364.996} C_VEL
LIN {X 0,Y 140.862,Z 1180.974,A -85,B 0,C 180,E1 30373.473,E2 30373.473} C_VEL
LIN {X 0,Y 145.967,Z 1177.769,A -85,B 0,C 180,E1 30380.052,E2 30380.052} C_VEL
LIN {X 0,Y 152.552,Z 1173.84,A -85,B 0,C 180,E1 30386.124,E2 30386.124} C_VEL
LIN {X 0,Y 189.926,Z 1156.266,A -85,B 0,C 180,E1 30398.858,E2 30398.858} C_VEL
LIN {X 0,Y 230.09,Z 1133.163,A -85,B 0,C 180,E1 30406.899,E2 30406.899} C_VEL
LIN {X 0,Y 268.697,Z 1106.31,A -85,B 0,C 180,E1 30412.067,E2 30412.067} C_VEL
LIN {X 0,Y 306.846,Z 1073.555,A -85,B 0,C 180,E1 30415.781,E2 30415.781} C_VEL
LIN {X 0,Y 312.876,Z 1067.87,A -85,B 0,C 180,E1 30416.341,E2 30416.341} C_VEL
LIN {X 0,Y 315.009,Z 1065.74,A -85,B 0,C 180,E1 30420.016,E2 30420.016} C_VEL
LIN {X 0,Y 314.284,Z 1067.113,A -85,B 0,C 180,E1 30422.212,E2 30422.212} C_VEL
LIN {X 0,Y 311.796,Z 1069.743,A -85,B 0,C 180,E1 30422.661,E2 30422.661} C_VEL
LIN {X 0,Y 273.536,Z 1103.964,A -85,B 0,C 180,E1 30426.06,E2 30426.06} C_VEL
LIN {X 0,Y 234.803,Z 1132.648,A -85,B 0,C 180,E1 30430.903,E2 30430.903} C_VEL
LIN {X 0,Y 194.128,Z 1157.39,A -85,B 0,C 180,E1 30438.478,E2 30438.478} C_VEL
LIN {X 0,Y 160.042,Z 1175.046,A -85,B 0,C 180,E1 30448.814,E2 30448.814} C_VEL
LIN {X 0,Y 130.172,Z 1188.699,A -85,B 0,C 180,E1 30465.847,E2 30465.847} C_VEL
LIN {X 0,Y 114.737,Z 1196.228,A -85,B 0,C 180,E1 30487.304,E2 30487.304} C_VEL
LIN {X 0,Y 111.879,Z 1198.317,A -85,B 0,C 180,E1 30502.234,E2 30502.234} C_VEL
LIN {X 0,Y 112.225,Z 1198.699,A -85,B 0,C 180,E1 30509.996,E2 30509.996} C_VEL
LIN {X 0,Y 112.694,Z 1197.46,A -85,B 0,C 180,E1 30525.552,E2 30525.552} C_VEL
LIN {X 0,Y 123.681,Z 1191.761,A -85,B 0,C 180,E1 30547.649,E2 30547.649} C_VEL
LIN {X 0,Y 147.054,Z 1181.213,A -85,B 0,C 180,E1 30565.288,E2 30565.288} C_VEL
LIN {X 0,Y 183.37,Z 1163.295,A -85,B 0,C 180,E1 30578.821,E2 30578.821} C_VEL
LIN {X 0,Y 222.73,Z 1140.593,A -85,B 0,C 180,E1 30587.222,E2 30587.222} C_VEL
LIN {X 0,Y 264.589,Z 1111.287,A -85,B 0,C 180,E1 30592.965,E2 30592.965} C_VEL
LIN {X 0,Y 300.902,Z 1080.434,A -85,B 0,C 180,E1 30596.452,E2 30596.452} C_VEL
LIN {X 0,Y 314.331,Z 1067.377,A -85,B 0,C 180,E1 30597.691,E2 30597.691} C_VEL
LIN {X 0,Y 315.085,Z 1065.946,A -85,B 0,C 180,E1 30599.984,E2 30599.984} C_VEL
LIN {X 0,Y 312.439,Z 1068.561,A -85,B 0,C 180,E1 30603.695,E2 30603.695} C_VEL
LIN {X 0,Y 274.187,Z 1102.108,A -85,B 0,C 180,E1 30607.254,E2 30607.254} C_VEL
LIN {X 0,Y 235.716,Z 1129.79,A -85,B 0,C 180,E1 30612.149,E2 30612.149} C_VEL
LIN {X 0,Y 196.356,Z 1152.893,A -85,B 0,C 180,E1 30619.491,E2 30619.491} C_VEL
LIN {X 0,Y 161.381,Z 1170.112,A -85,B 0,C 180,E1 30629.993,E2 30629.993} C_VEL
LIN {X 0,Y 131.769,Z 1182.556,A -85,B 0,C 180,E1 30646.527,E2 30646.527} C_VEL
LIN {X 0,Y 115.797,Z 1189.169,A -85,B 0,C 180,E1 30666.957,E2 30666.957} C_VEL
LIN {X 0,Y 112.114,Z 1191.039,A -85,B 0,C 180,E1 30682.258,E2 30682.258} C_VEL
LIN {X 0,Y 112.246,Z 1191.331,A -85,B 0,C 180,E1 30690.004,E2 30690.004} C_VEL
LIN {X 0,Y 113.294,Z 1190.292,A -85,B 0,C 180,E1 30705.476,E2 30705.476} C_VEL
LIN {X 0,Y 125.197,Z 1185.223,A -85,B 0,C 180,E1 30727.125,E2 30727.125} C_VEL
LIN {X 0,Y 148.844,Z 1175.527,A -85,B 0,C 180,E1 30744.315,E2 30744.315} C_VEL
LIN {X 0,Y 152.552,Z 1173.84,A -85,B 0,C 180,E1 30746.124,E2 30746.124} C_VEL
LIN {X 0,Y 160.506,Z 1169.64,A -85,B 0,C 180,E1 30751.624,E2 30751.624} C_VEL
LIN {X 0,Y 169.623,Z 1164.837,A -85,B 0,C 180,E1 30756.575,E2 30756.575} C_VEL
LIN {X 0,Y 207.498,Z 1145.711,A -85,B 0,C 180,E1 30765.448,E2 30765.448} C_VEL
LIN {X 0,Y 248.243,Z 1120.537,A -85,B 0,C 180,E1 30771.573,E2 30771.573} C_VEL
LIN {X 0,Y 286.272,Z 1091.673,A -85,B 0,C 180,E1 30775.593,E2 30775.593} C_VEL
LIN {X 0,Y 307.787,Z 1072.487,A -85,B 0,C 180,E1 30777.555,E2 30777.555} C_VEL
LIN {X 0,Y 309.261,Z 1071.301,A -85,B 0,C 180,E1 30780.016,E2 30780.016} C_VEL
LIN {X 0,Y 308.791,Z 1072.026,A -85,B 0,C 180,E1 30781.252,E2 30781.252} C_VEL
LIN {X 0,Y 270.386,Z 1105.633,A -85,B 0,C 180,E1 30784.572,E2 30784.572} C_VEL
LIN {X 0,Y 230.798,Z 1133.993,A -85,B 0,C 180,E1 30789.25,E2 30789.25} C_VEL
LIN {X 0,Y 189.267,Z 1158.422,A -85,B 0,C 180,E1 30796.64,E2 30796.64} C_VEL
LIN {X 0,Y 153.103,Z 1176.123,A -85,B 0,C 180,E1 30807.334,E2 30807.334} C_VEL
LIN {X 0,Y 124.394,Z 1188.428,A -85,B 0,C 180,E1 30823.203,E2 30823.203} C_VEL
LIN {X 0,Y 107.499,Z 1195.831,A -85,B 0,C 180,E1 30845.053,E2 30845.053} C_VEL
LIN {X 0,Y 103.978,Z 1198.055,A -85,B 0,C 180,E1 30861.639,E2 30861.639} C_VEL
LIN {X 0,Y 104.319,Z 1198.44,A -85,B 0,C 180,E1 30869.996,E2 30869.996} C_VEL
LIN {X 0,Y 104.987,Z 1197.197,A -85,B 0,C 180,E1 30886.726,E2 30886.726} C_VEL
LIN {X 0,Y 117.3,Z 1191.493,A -85,B 0,C 180,E1 30910.095,E2 30910.095} C_VEL
LIN {X 0,Y 142.493,Z 1180.942,A -85,B 0,C 180,E1 30928.03,E2 30928.03} C_VEL
LIN {X 0,Y 179.703,Z 1163.436,A -85,B 0,C 180,E1 30941.079,E2 30941.079} C_VEL
LIN {X 0,Y 219.317,Z 1141.428,A -85,B 0,C 180,E1 30949.052,E2 30949.052} C_VEL
LIN {X 0,Y 260.687,Z 1113.256,A -85,B 0,C 180,E1 30954.431,E2 30954.431} C_VEL
LIN {X 0,Y 298.644,Z 1081.939,A -85,B 0,C 180,E1 30957.867,E2 30957.867} C_VEL
LIN {X 0,Y 308.868,Z 1072.208,A -85,B 0,C 180,E1 30958.746,E2 30958.746} C_VEL
LIN {X 0,Y 309.325,Z 1071.5,A -85,B 0,C 180,E1 30959.984,E2 30959.984} C_VEL
LIN {X 0,Y 307.839,Z 1072.705,A -85,B 0,C 180,E1 30962.445,E2 30962.445} C_VEL
LIN {X 0,Y 269.126,Z 1105.659,A -85,B 0,C 180,E1 30965.979,E2 30965.979} C_VEL
LIN {X 0,Y 230.656,Z 1132.179,A -85,B 0,C 180,E1 30970.682,E2 30970.682} C_VEL
LIN {X 0,Y 190.558,Z 1154.853,A -85,B 0,C 180,E1 30977.908,E2 30977.908} C_VEL
LIN {X 0,Y 154.66,Z 1171.488,A -85,B 0,C 180,E1 30988.442,E2 30988.442} C_VEL
LIN {X 0,Y 122.851,Z 1184.044,A -85,B 0,C 180,E1 31006.557,E2 31006.557} C_VEL
LIN {X 0,Y 108.446,Z 1189.432,A -85,B 0,C 180,E1 31025.294,E2 31025.294} C_VEL
LIN {X 0,Y 104.246,Z 1191.3,A -85,B 0,C 180,E1 31041.669,E2 31041.669} C_VEL
LIN {X 0,Y 104.338,Z 1191.591,A -85,B 0,C 180,E1 31050.004,E2 31050.004} C_VEL
LIN {X 0,Y 105.602,Z 1190.555,A -85,B 0,C 180,E1 31066.634,E2 31066.634} C_VEL
LIN {X 0,Y 118.807,Z 1185.491,A -85,B 0,C 180,E1 31089.495,E2 31089.495} C_VEL
LIN {X 0,Y 146.686,Z 1174.728,A -85,B 0,C 180,E1 31108.112,E2 31108.112} C_VEL
LIN {X 0,Y 169.623,Z 1164.837,A -85,B 0,C 180,E1 31116.575,E2 31116.575} C_VEL
LIN {X 0,Y 179.725,Z 1159.686,A -85,B 0,C 180,E1 31120.967,E2 31120.967} C_VEL
LIN {X 0,Y 190.456,Z 1153.84,A -85,B 0,C 180,E1 31124.871,E2 31124.871} C_VEL
LIN {X 0,Y 232.399,Z 1130.419,A -85,B 0,C 180,E1 31131.686,E2 31131.686} C_VEL
LIN {X 0,Y 272.645,Z 1102.39,A -85,B 0,C 180,E1 31136.08,E2 31136.08} C_VEL
LIN {X 0,Y 302.329,Z 1077.551,A -85,B 0,C 180,E1 31138.531,E2 31138.531} C_VEL
LIN {X 0,Y 303.396,Z 1076.731,A -85,B 0,C 180,E1 31140.017,E2 31140.017} C_VEL
LIN {X 0,Y 292.828,Z 1086.347,A -85,B 0,C 180,E1 31140.977,E2 31140.977} C_VEL
LIN {X 0,Y 252.371,Z 1118.421,A -85,B 0,C 180,E1 31144.549,E2 31144.549} C_VEL
LIN {X 0,Y 211.512,Z 1144.713,A -85,B 0,C 180,E1 31149.788,E2 31149.788} C_VEL
LIN {X 0,Y 168.667,Z 1167.256,A -85,B 0,C 180,E1 31158.512,E2 31158.512} C_VEL
LIN {X 0,Y 132.498,Z 1182.835,A -85,B 0,C 180,E1 31171.835,E2 31171.835} C_VEL
LIN {X 0,Y 106.819,Z 1192.858,A -85,B 0,C 180,E1 31192.071,E2 31192.071} C_VEL
LIN {X 0,Y 97.3,Z 1196.917,A -85,B 0,C 180,E1 31211.899,E2 31211.899} C_VEL
LIN {X 0,Y 96.387,Z 1198.18,A -85,B 0,C 180,E1 31229.996,E2 31229.996} C_VEL
LIN {X 0,Y 98.685,Z 1196.292,A -85,B 0,C 180,E1 31253.144,E2 31253.144} C_VEL
LIN {X 0,Y 114.85,Z 1189.844,A -85,B 0,C 180,E1 31276.351,E2 31276.351} C_VEL
LIN {X 0,Y 146.606,Z 1177.114,A -85,B 0,C 180,E1 31294.4,E2 31294.4} C_VEL
LIN {X 0,Y 183.74,Z 1160.016,A -85,B 0,C 180,E1 31305.083,E2 31305.083} C_VEL
LIN {X 0,Y 225.802,Z 1136.224,A -85,B 0,C 180,E1 31312.287,E2 31312.287} C_VEL
LIN {X 0,Y 265.686,Z 1108.848,A -85,B 0,C 180,E1 31316.782,E2 31316.782} C_VEL
LIN {X 0,Y 302.218,Z 1078.13,A -85,B 0,C 180,E1 31319.71,E2 31319.71} C_VEL
LIN {X 0,Y 303.463,Z 1076.927,A -85,B 0,C 180,E1 31319.983,E2 31319.983} C_VEL
LIN {X 0,Y 302.303,Z 1077.842,A -85,B 0,C 180,E1 31321.39,E2 31321.39} C_VEL
LIN {X 0,Y 265.2,Z 1108.31,A -85,B 0,C 180,E1 31324.553,E2 31324.553} C_VEL
LIN {X 0,Y 222.633,Z 1136.454,A -85,B 0,C 180,E1 31329.584,E2 31329.584} C_VEL
LIN {X 0,Y 183.803,Z 1157.292,A -85,B 0,C 180,E1 31336.477,E2 31336.477} C_VEL
LIN {X 0,Y 143.271,Z 1174.772,A -85,B 0,C 180,E1 31348.689,E2 31348.689} C_VEL
LIN {X 0,Y 112.574,Z 1185.819,A -85,B 0,C 180,E1 31367.848,E2 31367.848} C_VEL
LIN {X 0,Y 97.927,Z 1190.844,A -85,B 0,C 180,E1 31392.029,E2 31392.029} C_VEL
LIN {X 0,Y 96.419,Z 1191.851,A -85,B 0,C 180,E1 31410.004,E2 31410.004} C_VEL
LIN {X 0,Y 97.953,Z 1190.818,A -85,B 0,C 180,E1 31427.976,E2 31427.976} C_VEL
LIN {X 0,Y 112.663,Z 1185.758,A -85,B 0,C 180,E1 31452.121,E2 31452.121} C_VEL
LIN {X 0,Y 139.907,Z 1176.068,A -85,B 0,C 180,E1 31469.783,E2 31469.783} C_VEL
LIN {X 0,Y 179.361,Z 1159.224,A -85,B 0,C 180,E1 31482.449,E2 31482.449} C_VEL
LIN {X 0,Y 190.456,Z 1153.84,A -85,B 0,C 180,E1 31484.871,E2 31484.871} C_VEL
LIN {X 0,Y 201.808,Z 1147.732,A -85,B 0,C 180,E1 31488.337,E2 31488.337} C_VEL
LIN {X 0,Y 213.692,Z 1141,A -85,B 0,C 180,E1 31491.396,E2 31491.396} C_VEL
LIN {X 0,Y 253.706,Z 1116.108,A -85,B 0,C 180,E1 31496.101,E2 31496.101} C_VEL
LIN {X 0,Y 292.542,Z 1086.297,A -85,B 0,C 180,E1 31499.377,E2 31499.377} C_VEL
LIN {X 0,Y 251.501,Z 1118.396,A -85,B 0,C 180,E1 31502.688,E2 31502.688} C_VEL
LIN {X 0,Y 210.502,Z 1144.29,A -85,B 0,C 180,E1 31507.49,E2 31507.49} C_VEL
LIN {X 0,Y 165.729,Z 1167.212,A -85,B 0,C 180,E1 31515.904,E2 31515.904} C_VEL
LIN {X 0,Y 126.999,Z 1183.048,A -85,B 0,C 180,E1 31529.32,E2 31529.32} C_VEL
LIN {X 0,Y 101.136,Z 1192.338,A -85,B 0,C 180,E1 31548.404,E2 31548.404} C_VEL
LIN {X 0,Y 89.684,Z 1196.652,A -85,B 0,C 180,E1 31570.302,E2 31570.302} C_VEL
LIN {X 0,Y 88.475,Z 1197.92,A -85,B 0,C 180,E1 31589.995,E2 31589.995} C_VEL
LIN {X 0,Y 89.679,Z 1196.668,A -85,B 0,C 180,E1 31609.689,E2 31609.689} C_VEL
LIN {X 0,Y 105.255,Z 1190.954,A -85,B 0,C 180,E1 31635.87,E2 31635.87} C_VEL
LIN {X 0,Y 134.43,Z 1180.398,A -85,B 0,C 180,E1 31654.054,E2 31654.054} C_VEL
LIN {X 0,Y 175.01,Z 1162.892,A -85,B 0,C 180,E1 31666.248,E2 31666.248} C_VEL
LIN {X 0,Y 215.858,Z 1141.436,A -85,B 0,C 180,E1 31673.242,E2 31673.242} C_VEL
LIN {X 0,Y 258.932,Z 1113.201,A -85,B 0,C 180,E1 31678.014,E2 31678.014} C_VEL
LIN {X 0,Y 291.88,Z 1087.1,A -85,B 0,C 180,E1 31680.578,E2 31680.578} C_VEL
LIN {X 0,Y 251.831,Z 1117.633,A -85,B 0,C 180,E1 31684.008,E2 31684.008} C_VEL
LIN {X 0,Y 210.359,Z 1142.929,A -85,B 0,C 180,E1 31688.998,E2 31688.998} C_VEL
LIN {X 0,Y 169.512,Z 1163.011,A -85,B 0,C 180,E1 31696.612,E2 31696.612} C_VEL
LIN {X 0,Y 135.894,Z 1176.443,A -85,B 0,C 180,E1 31707.186,E2 31707.186} C_VEL
LIN {X 0,Y 106.388,Z 1186.169,A -85,B 0,C 180,E1 31725.176,E2 31725.176} C_VEL
LIN {X 0,Y 90.358,Z 1191.106,A -85,B 0,C 180,E1 31750.465,E2 31750.465} C_VEL
LIN {X 0,Y 88.498,Z 1192.111,A -85,B 0,C 180,E1 31770.005,E2 31770.005} C_VEL
LIN {X 0,Y 90.383,Z 1191.081,A -85,B 0,C 180,E1 31789.54,E2 31789.54} C_VEL
LIN {X 0,Y 106.76,Z 1186.026,A -85,B 0,C 180,E1 31815.055,E2 31815.055} C_VEL
LIN {X 0,Y 135.964,Z 1176.338,A -85,B 0,C 180,E1 31832.771,E2 31832.771} C_VEL
LIN {X 0,Y 175.793,Z 1160.061,A -85,B 0,C 180,E1 31844.716,E2 31844.716} C_VEL
LIN {X 0,Y 213.692,Z 1141,A -85,B 0,C 180,E1 31851.396,E2 31851.396} C_VEL
LIN {X 0,Y 225.888,Z 1133.948,A -85,B 0,C 180,E1 31854.134,E2 31854.134} C_VEL
LIN {X 0,Y 236.544,Z 1127.28,A -85,B 0,C 180,E1 31856.317,E2 31856.317} C_VEL
LIN {X 0,Y 238.269,Z 1126.174,A -85,B 0,C 180,E1 31856.504,E2 31856.504} C_VEL
LIN {X 0,Y 268.022,Z 1105.973,A -85,B 0,C 180,E1 31859.188,E2 31859.188} C_VEL
LIN {X 0,Y 259.326,Z 1112.346,A -85,B 0,C 180,E1 31860.107,E2 31860.107} C_VEL
LIN {X 0,Y 216.184,Z 1140.344,A -85,B 0,C 180,E1 31864.419,E2 31864.419} C_VEL
LIN {X 0,Y 172.516,Z 1162.831,A -85,B 0,C 180,E1 31871.192,E2 31871.192} C_VEL
LIN {X 0,Y 131.002,Z 1180.049,A -85,B 0,C 180,E1 31882.652,E2 31882.652} C_VEL
LIN {X 0,Y 99.676,Z 1190.643,A -85,B 0,C 180,E1 31900.704,E2 31900.704} C_VEL
LIN {X 0,Y 82.127,Z 1196.387,A -85,B 0,C 180,E1 31928.402,E2 31928.402} C_VEL
LIN {X 0,Y 80.536,Z 1197.659,A -85,B 0,C 180,E1 31949.995,E2 31949.995} C_VEL
LIN {X 0,Y 82.803,Z 1196.142,A -85,B 0,C 180,E1 31974.019,E2 31974.019} C_VEL
LIN {X 0,Y 99.688,Z 1190.684,A -85,B 0,C 180,E1 31999.275,E2 31999.275} C_VEL
LIN {X 0,Y 133.973,Z 1178.965,A -85,B 0,C 180,E1 32018.423,E2 32018.423} C_VEL
LIN {X 0,Y 178.125,Z 1160.393,A -85,B 0,C 180,E1 32029.849,E2 32029.849} C_VEL
LIN {X 0,Y 220.136,Z 1138.109,A -85,B 0,C 180,E1 32036.042,E2 32036.042} C_VEL
LIN {X 0,Y 264.136,Z 1109.119,A -85,B 0,C 180,E1 32040.249,E2 32040.249} C_VEL
LIN {X 0,Y 267.452,Z 1106.634,A -85,B 0,C 180,E1 32040.779,E2 32040.779} C_VEL
LIN {X 0,Y 227.378,Z 1132.984,A -85,B 0,C 180,E1 32044.557,E2 32044.557} C_VEL
LIN {X 0,Y 184.457,Z 1155.661,A -85,B 0,C 180,E1 32050.572,E2 32050.572} C_VEL
LIN {X 0,Y 144.551,Z 1172.295,A -85,B 0,C 180,E1 32059.815,E2 32059.815} C_VEL
LIN {X 0,Y 110.386,Z 1183.625,A -85,B 0,C 180,E1 32074.786,E2 32074.786} C_VEL
LIN {X 0,Y 87.067,Z 1190.225,A -85,B 0,C 180,E1 32098.629,E2 32098.629} C_VEL
LIN {X 0,Y 80.691,Z 1192.083,A -85,B 0,C 180,E1 32119.212,E2 32119.212} C_VEL
LIN {X 0,Y 80.576,Z 1192.371,A -85,B 0,C 180,E1 32130.005,E2 32130.005} C_VEL
LIN {X 0,Y 85.249,Z 1190.758,A -85,B 0,C 180,E1 32157.729,E2 32157.729} C_VEL
LIN {X 0,Y 105.656,Z 1185.04,A -85,B 0,C 180,E1 32181.877,E2 32181.877} C_VEL
LIN {X 0,Y 140.764,Z 1173.552,A -85,B 0,C 180,E1 32198.922,E2 32198.922} C_VEL
LIN {X 0,Y 180.665,Z 1157.357,A -85,B 0,C 180,E1 32208.647,E2 32208.647} C_VEL
LIN {X 0,Y 224.994,Z 1134.212,A -85,B 0,C 180,E1 32215.088,E2 32215.088} C_VEL
LIN {X 0,Y 238.269,Z 1126.174,A -85,B 0,C 180,E1 32216.504,E2 32216.504} C_VEL
LIN {X 0,Y 238.868,Z 1125.814,A -85,B 0,C 180,E1 32217.386,E2 32217.386} C_VEL
LIN {X 0,Y 234.062,Z 1128.948,A -85,B 0,C 180,E1 32219.172,E2 32219.172} C_VEL
LIN {X 0,Y 221.143,Z 1136.831,A -85,B 0,C 180,E1 32221.547,E2 32221.547} C_VEL
LIN {X 0,Y 216.431,Z 1139.638,A -85,B 0,C 180,E1 32222.141,E2 32222.141} C_VEL
LIN {X 0,Y 173.501,Z 1161.49,A -85,B 0,C 180,E1 32228.039,E2 32228.039} C_VEL
LIN {X 0,Y 128.036,Z 1179.776,A -85,B 0,C 180,E1 32239.224,E2 32239.224} C_VEL
LIN {X 0,Y 94.501,Z 1190.372,A -85,B 0,C 180,E1 32256.908,E2 32256.908} C_VEL
LIN {X 0,Y 74.689,Z 1196.122,A -85,B 0,C 180,E1 32286.125,E2 32286.125} C_VEL
LIN {X 0,Y 72.605,Z 1197.399,A -85,B 0,C 180,E1 32309.994,E2 32309.994} C_VEL
LIN {X 0,Y 74.683,Z 1196.139,A -85,B 0,C 180,E1 32333.864,E2 32333.864} C_VEL
LIN {X 0,Y 94.512,Z 1190.414,A -85,B 0,C 180,E1 32363.068,E2 32363.068} C_VEL
LIN {X 0,Y 130.975,Z 1178.758,A -85,B 0,C 180,E1 32381.742,E2 32381.742} C_VEL
LIN {X 0,Y 176.186,Z 1160.411,A -85,B 0,C 180,E1 32392.402,E2 32392.402} C_VEL
LIN {X 0,Y 219.719,Z 1137.838,A -85,B 0,C 180,E1 32398.206,E2 32398.206} C_VEL
LIN {X 0,Y 246.325,Z 1121.347,A -85,B 0,C 180,E1 32400.673,E2 32400.673} C_VEL
LIN {X 0,Y 201.129,Z 1147.266,A -85,B 0,C 180,E1 32405.466,E2 32405.466} C_VEL
LIN {X 0,Y 158.678,Z 1166.302,A -85,B 0,C 180,E1 32412.558,E2 32412.558} C_VEL
LIN {X 0,Y 117.118,Z 1180.687,A -85,B 0,C 180,E1 32425.43,E2 32425.43} C_VEL
LIN {X 0,Y 87.243,Z 1188.882,A -85,B 0,C 180,E1 32446.152,E2 32446.152} C_VEL
LIN {X 0,Y 72.876,Z 1192.345,A -85,B 0,C 180,E1 32478.039,E2 32478.039} C_VEL
LIN {X 0,Y 72.652,Z 1192.631,A -85,B 0,C 180,E1 32490.006,E2 32490.006} C_VEL
LIN {X 0,Y 75.463,Z 1191.607,A -85,B 0,C 180,E1 32513.615,E2 32513.615} C_VEL
LIN {X 0,Y 95.934,Z 1186.562,A -85,B 0,C 180,E1 32541.967,E2 32541.967} C_VEL
LIN {X 0,Y 130.661,Z 1176.387,A -85,B 0,C 180,E1 32559.743,E2 32559.743} C_VEL
LIN {X 0,Y 176.809,Z 1158.647,A -85,B 0,C 180,E1 32570.825,E2 32570.825} C_VEL
LIN {X 0,Y 219.552,Z 1137.286,A -85,B 0,C 180,E1 32576.645,E2 32576.645} C_VEL
LIN {X 0,Y 246.733,Z 1120.907,A -85,B 0,C 180,E1 32579.277,E2 32579.277} C_VEL
LIN {X 0,Y 216.431,Z 1139.638,A -85,B 0,C 180,E1 32582.141,E2 32582.141} C_VEL
LIN {X 0,Y 201.054,Z 1147.808,A -85,B 0,C 180,E1 32582.728,E2 32582.728} C_VEL
LIN {X 0,Y 185.377,Z 1155.303,A -85,B 0,C 180,E1 32583.441,E2 32583.441} C_VEL
LIN {X 0,Y 142.423,Z 1173.552,A -85,B 0,C 180,E1 32591.045,E2 32591.045} C_VEL
LIN {X 0,Y 100.716,Z 1187.069,A -85,B 0,C 180,E1 32605.803,E2 32605.803} C_VEL
LIN {X 0,Y 72.678,Z 1194.494,A -85,B 0,C 180,E1 32631.402,E2 32631.402} C_VEL
LIN {X 0,Y 64.683,Z 1196.742,A -85,B 0,C 180,E1 32656.483,E2 32656.483} C_VEL
LIN {X 0,Y 64.66,Z 1197.138,A -85,B 0,C 180,E1 32669.993,E2 32669.993} C_VEL
LIN {X 0,Y 67.391,Z 1195.875,A -85,B 0,C 180,E1 32696.638,E2 32696.638} C_VEL
LIN {X 0,Y 89.8,Z 1190.144,A -85,B 0,C 180,E1 32727.277,E2 32727.277} C_VEL
LIN {X 0,Y 125.542,Z 1179.583,A -85,B 0,C 180,E1 32744.339,E2 32744.339} C_VEL
LIN {X 0,Y 170.883,Z 1162.042,A -85,B 0,C 180,E1 32754.422,E2 32754.422} C_VEL
LIN {X 0,Y 215.574,Z 1139.931,A -85,B 0,C 180,E1 32759.977,E2 32759.977} C_VEL
LIN {X 0,Y 220.31,Z 1137.163,A -85,B 0,C 180,E1 32760.43,E2 32760.43} C_VEL
LIN {X 0,Y 221.52,Z 1136.422,A -85,B 0,C 180,E1 32760.898,E2 32760.898} C_VEL
LIN {X 0,Y 178.528,Z 1157.861,A -85,B 0,C 180,E1 32766.006,E2 32766.006} C_VEL
LIN {X 0,Y 133.107,Z 1175.044,A -85,B 0,C 180,E1 32775.222,E2 32775.222} C_VEL
LIN {X 0,Y 96.351,Z 1185.651,A -85,B 0,C 180,E1 32790.401,E2 32790.401} C_VEL
LIN {X 0,Y 73.758,Z 1190.754,A -85,B 0,C 180,E1 32812.083,E2 32812.083} C_VEL
LIN {X 0,Y 65.097,Z 1192.607,A -85,B 0,C 180,E1 32836.584,E2 32836.584} C_VEL
LIN {X 0,Y 64.726,Z 1192.891,A -85,B 0,C 180,E1 32850.007,E2 32850.007} C_VEL
LIN {X 0,Y 69.416,Z 1191.619,A -85,B 0,C 180,E1 32879.613,E2 32879.613} C_VEL
LIN {X 0,Y 91.134,Z 1186.83,A -85,B 0,C 180,E1 32906.011,E2 32906.011} C_VEL
LIN {X 0,Y 126.591,Z 1177.151,A -85,B 0,C 180,E1 32922.749,E2 32922.749} C_VEL
LIN {X 0,Y 170.282,Z 1161.153,A -85,B 0,C 180,E1 32932.61,E2 32932.61} C_VEL
LIN {X 0,Y 214.948,Z 1139.981,A -85,B 0,C 180,E1 32938.347,E2 32938.347} C_VEL
LIN {X 0,Y 222.081,Z 1135.942,A -85,B 0,C 180,E1 32939.071,E2 32939.071} C_VEL
LIN {X 0,Y 217.487,Z 1138.657,A -85,B 0,C 180,E1 32939.818,E2 32939.818} C_VEL
LIN {X 0,Y 185.377,Z 1155.303,A -85,B 0,C 180,E1 32943.441,E2 32943.441} C_VEL
LIN {X 0,Y 169.47,Z 1162.289,A -85,B 0,C 180,E1 32944.283,E2 32944.283} C_VEL
LIN {X 0,Y 153.409,Z 1168.563,A -85,B 0,C 180,E1 32945.387,E2 32945.387} C_VEL
LIN {X 0,Y 110.114,Z 1183.265,A -85,B 0,C 180,E1 32956.119,E2 32956.119} C_VEL
LIN {X 0,Y 73.626,Z 1192.687,A -85,B 0,C 180,E1 32978.086,E2 32978.086} C_VEL
LIN {X 0,Y 56.924,Z 1196.479,A -85,B 0,C 180,E1 33014.598,E2 33014.598} C_VEL
LIN {X 0,Y 56.711,Z 1196.877,A -85,B 0,C 180,E1 33029.992,E2 33029.992} C_VEL
LIN {X 0,Y 60.261,Z 1195.609,A -85,B 0,C 180,E1 33060.092,E2 33060.092} C_VEL
LIN {X 0,Y 80.223,Z 1191.155,A -85,B 0,C 180,E1 33087.945,E2 33087.945} C_VEL
LIN {X 0,Y 120.158,Z 1180.324,A -85,B 0,C 180,E1 33107.094,E2 33107.094} C_VEL
LIN {X 0,Y 162.808,Z 1164.953,A -85,B 0,C 180,E1 33116.13,E2 33116.13} C_VEL
LIN {X 0,Y 199.977,Z 1147.936,A -85,B 0,C 180,E1 33120.764,E2 33120.764} C_VEL
LIN {X 0,Y 155.462,Z 1167.008,A -85,B 0,C 180,E1 33126.736,E2 33126.736} C_VEL
LIN {X 0,Y 111.066,Z 1181.224,A -85,B 0,C 180,E1 33137.765,E2 33137.765} C_VEL
LIN {X 0,Y 76.352,Z 1189.415,A -85,B 0,C 180,E1 33157.668,E2 33157.668} C_VEL
LIN {X 0,Y 57.369,Z 1192.868,A -85,B 0,C 180,E1 33194.736,E2 33194.736} C_VEL
LIN {X 0,Y 56.798,Z 1193.151,A -85,B 0,C 180,E1 33210.008,E2 33210.008} C_VEL
LIN {X 0,Y 61.103,Z 1192.134,A -85,B 0,C 180,E1 33239.652,E2 33239.652} C_VEL
LIN {X 0,Y 86.842,Z 1187.098,A -85,B 0,C 180,E1 33270.472,E2 33270.472} C_VEL
LIN {X 0,Y 124.404,Z 1177.421,A -85,B 0,C 180,E1 33286.362,E2 33286.362} C_VEL
LIN {X 0,Y 170.525,Z 1160.976,A -85,B 0,C 180,E1 33295.535,E2 33295.535} C_VEL
LIN {X 0,Y 200.37,Z 1147.592,A -85,B 0,C 180,E1 33299.192,E2 33299.192} C_VEL
LIN {X 0,Y 155.492,Z 1167.772,A -85,B 0,C 180,E1 33305.016,E2 33305.016} C_VEL
LIN {X 0,Y 153.409,Z 1168.563,A -85,B 0,C 180,E1 33305.387,E2 33305.387} C_VEL
LIN {X 0,Y 145.505,Z 1171.48,A -85,B 0,C 180,E1 33306.315,E2 33306.315} C_VEL
LIN {X 0,Y 122.717,Z 1178.769,A -85,B 0,C 180,E1 33307.971,E2 33307.971} C_VEL
LIN {X 0,Y 120.796,Z 1179.333,A -85,B 0,C 180,E1 33308.394,E2 33308.394} C_VEL
LIN {X 0,Y 76.172,Z 1190.84,A -85,B 0,C 180,E1 33326.77,E2 33326.77} C_VEL
LIN {X 0,Y 53.421,Z 1195.325,A -85,B 0,C 180,E1 33355.536,E2 33355.536} C_VEL
LIN {X 0,Y 48.758,Z 1196.616,A -85,B 0,C 180,E1 33389.991,E2 33389.991} C_VEL
LIN {X 0,Y 53.414,Z 1195.344,A -85,B 0,C 180,E1 33424.449,E2 33424.449} C_VEL
LIN {X 0,Y 82.059,Z 1189.603,A -85,B 0,C 180,E1 33457.022,E2 33457.022} C_VEL
LIN {X 0,Y 122.102,Z 1179.037,A -85,B 0,C 180,E1 33471.89,E2 33471.89} C_VEL
LIN {X 0,Y 171.545,Z 1160.884,A -85,B 0,C 180,E1 33480.207,E2 33480.207} C_VEL
LIN {X 0,Y 175.297,Z 1159.296,A -85,B 0,C 180,E1 33480.978,E2 33480.978} C_VEL
LIN {X 0,Y 126.209,Z 1176.687,A -85,B 0,C 180,E1 33488.987,E2 33488.987} C_VEL
LIN {X 0,Y 83.062,Z 1187.422,A -85,B 0,C 180,E1 33504.558,E2 33504.558} C_VEL
LIN {X 0,Y 53.912,Z 1192.476,A -85,B 0,C 180,E1 33537.051,E2 33537.051} C_VEL
LIN {X 0,Y 48.867,Z 1193.412,A -85,B 0,C 180,E1 33570.009,E2 33570.009} C_VEL
LIN {X 0,Y 54.273,Z 1192.398,A -85,B 0,C 180,E1 33603.848,E2 33603.848} C_VEL
LIN {X 0,Y 83.121,Z 1187.367,A -85,B 0,C 180,E1 33635.377,E2 33635.377} C_VEL
LIN {X 0,Y 126.244,Z 1176.588,A -85,B 0,C 180,E1 33650.954,E2 33650.954} C_VEL
LIN {X 0,Y 175.695,Z 1159.02,A -85,B 0,C 180,E1 33658.986,E2 33658.986} C_VEL
LIN {X 0,Y 147.196,Z 1170.39,A -85,B 0,C 180,E1 33663.159,E2 33663.159} C_VEL
LIN {X 0,Y 120.796,Z 1179.333,A -85,B 0,C 180,E1 33668.394,E2 33668.394} C_VEL
LIN {X 0,Y 104.369,Z 1183.709,A -85,B 0,C 180,E1 33670.638,E2 33670.638} C_VEL
LIN {X 0,Y 87.922,Z 1187.382,A -85,B 0,C 180,E1 33673.582,E2 33673.582} C_VEL
LIN {X 0,Y 55.696,Z 1193.69,A -85,B 0,C 180,E1 33695.504,E2 33695.504} C_VEL
LIN {X 0,Y 41.687,Z 1195.953,A -85,B 0,C 180,E1 33728.736,E2 33728.736} C_VEL
LIN {X 0,Y 40.816,Z 1196.356,A -85,B 0,C 180,E1 33749.989,E2 33749.989} C_VEL
LIN {X 0,Y 46.953,Z 1195.078,A -85,B 0,C 180,E1 33790.054,E2 33790.054} C_VEL
LIN {X 0,Y 79.205,Z 1189.333,A -85,B 0,C 180,E1 33822.52,E2 33822.52} C_VEL
LIN {X 0,Y 121.208,Z 1178.765,A -85,B 0,C 180,E1 33835.795,E2 33835.795} C_VEL
LIN {X 0,Y 151.113,Z 1168.708,A -85,B 0,C 180,E1 33840.645,E2 33840.645} C_VEL
LIN {X 0,Y 151.131,Z 1168.669,A -85,B 0,C 180,E1 33841.095,E2 33841.095} C_VEL
LIN {X 0,Y 107.202,Z 1181.761,A -85,B 0,C 180,E1 33849.375,E2 33849.375} C_VEL
LIN {X 0,Y 67.661,Z 1189.947,A -85,B 0,C 180,E1 33866.717,E2 33866.717} C_VEL
LIN {X 0,Y 42.181,Z 1193.392,A -85,B 0,C 180,E1 33909.018,E2 33909.018} C_VEL
LIN {X 0,Y 40.934,Z 1193.672,A -85,B 0,C 180,E1 33930.011,E2 33930.011} C_VEL
LIN {X 0,Y 47.804,Z 1192.662,A -85,B 0,C 180,E1 33969.225,E2 33969.225} C_VEL
LIN {X 0,Y 80.068,Z 1187.635,A -85,B 0,C 180,E1 34000.688,E2 34000.688} C_VEL
LIN {X 0,Y 125.217,Z 1176.859,A -85,B 0,C 180,E1 34014.663,E2 34014.663} C_VEL
LIN {X 0,Y 151.15,Z 1168.557,A -85,B 0,C 180,E1 34018.84,E2 34018.84} C_VEL
LIN {X 0,Y 151.129,Z 1168.601,A -85,B 0,C 180,E1 34019.342,E2 34019.342} C_VEL
LIN {X 0,Y 103.249,Z 1183.69,A -85,B 0,C 180,E1 34028.464,E2 34028.464} C_VEL
LIN {X 0,Y 87.922,Z 1187.382,A -85,B 0,C 180,E1 34033.582,E2 34033.582} C_VEL
LIN {X 0,Y 71.642,Z 1190.437,A -85,B 0,C 180,E1 34037.724,E2 34037.724} C_VEL
LIN {X 0,Y 55.643,Z 1192.75,A -85,B 0,C 180,E1 34044.057,E2 34044.057} C_VEL
LIN {X 0,Y 34.316,Z 1195.689,A -85,B 0,C 180,E1 34083.86,E2 34083.86} C_VEL
LIN {X 0,Y 32.854,Z 1196.094,A -85,B 0,C 180,E1 34109.987,E2 34109.987} C_VEL
LIN {X 0,Y 41.078,Z 1194.812,A -85,B 0,C 180,E1 34157.353,E2 34157.353} C_VEL
LIN {X 0,Y 78.084,Z 1188.885,A -85,B 0,C 180,E1 34188.777,E2 34188.777} C_VEL
LIN {X 0,Y 122.209,Z 1178.077,A -85,B 0,C 180,E1 34199.959,E2 34199.959} C_VEL
LIN {X 0,Y 127.992,Z 1176.255,A -85,B 0,C 180,E1 34200.99,E2 34200.99} C_VEL
LIN {X 0,Y 87.9,Z 1186.032,A -85,B 0,C 180,E1 34209.84,E2 34209.84} C_VEL
LIN {X 0,Y 52.173,Z 1191.815,A -85,B 0,C 180,E1 34229.686,E2 34229.686} C_VEL
LIN {X 0,Y 34.839,Z 1193.654,A -85,B 0,C 180,E1 34264.309,E2 34264.309} C_VEL
LIN {X 0,Y 32.998,Z 1193.933,A -85,B 0,C 180,E1 34290.013,E2 34290.013} C_VEL
LIN {X 0,Y 41.88,Z 1192.927,A -85,B 0,C 180,E1 34336.205,E2 34336.205} C_VEL
LIN {X 0,Y 77.75,Z 1187.904,A -85,B 0,C 180,E1 34366.38,E2 34366.38} C_VEL
LIN {X 0,Y 124.669,Z 1177.145,A -85,B 0,C 180,E1 34378.414,E2 34378.414} C_VEL
LIN {X 0,Y 128.366,Z 1176.054,A -85,B 0,C 180,E1 34378.983,E2 34378.983} C_VEL
LIN {X 0,Y 84.156,Z 1187.617,A -85,B 0,C 180,E1 34388.978,E2 34388.978} C_VEL
LIN {X 0,Y 55.643,Z 1192.75,A -85,B 0,C 180,E1 34404.057,E2 34404.057} C_VEL
LIN {X 0,Y 44.425,Z 1194.134,A -85,B 0,C 180,E1 34411.77,E2 34411.77} C_VEL
LIN {X 0,Y 28.62,Z 1195.345,A -85,B 0,C 180,E1 34431.167,E2 34431.167} C_VEL
LIN {X 0,Y 27.598,Z 1195.386,A -85,B 0,C 180,E1 34435.141,E2 34435.141} C_VEL
LIN {X 0,Y 24.912,Z 1195.833,A -85,B 0,C 180,E1 34469.983,E2 34469.983} C_VEL
LIN {X 0,Y 36.074,Z 1194.546,A -85,B 0,C 180,E1 34526.886,E2 34526.886} C_VEL
LIN {X 0,Y 75.897,Z 1188.791,A -85,B 0,C 180,E1 34554.505,E2 34554.505} C_VEL
LIN {X 0,Y 101.914,Z 1183.246,A -85,B 0,C 180,E1 34561.259,E2 34561.259} C_VEL
LIN {X 0,Y 58.81,Z 1190.859,A -85,B 0,C 180,E1 34574.799,E2 34574.799} C_VEL
LIN {X 0,Y 27.877,Z 1193.916,A -85,B 0,C 180,E1 34617.195,E2 34617.195} C_VEL
LIN {X 0,Y 25.068,Z 1194.193,A -85,B 0,C 180,E1 34650.017,E2 34650.017} C_VEL
LIN {X 0,Y 36.769,Z 1193.191,A -85,B 0,C 180,E1 34705.301,E2 34705.301} C_VEL
LIN {X 0,Y 76.241,Z 1188.172,A -85,B 0,C 180,E1 34732.354,E2 34732.354} C_VEL
LIN {X 0,Y 102.084,Z 1183.13,A -85,B 0,C 180,E1 34738.7,E2 34738.7} C_VEL
LIN {X 0,Y 75.907,Z 1188.743,A -85,B 0,C 180,E1 34745.459,E2 34745.459} C_VEL
LIN {X 0,Y 36.081,Z 1194.526,A -85,B 0,C 180,E1 34773.088,E2 34773.088} C_VEL
LIN {X 0,Y 27.598,Z 1195.386,A -85,B 0,C 180,E1 34795.141,E2 34795.141} C_VEL
LIN {X 0,Y 21.722,Z 1195.731,A -85,B 0,C 180,E1 34822.663,E2 34822.663} C_VEL
LIN {X 0,Y 23.296,Z 1194.961,A -85,B 0,C 180,E1 34883.046,E2 34883.046} C_VEL
LIN {X 0,Y 60.546,Z 1191.063,A -85,B 0,C 180,E1 34916.559,E2 34916.559} C_VEL
LIN {X 0,Y 75.57,Z 1188.494,A -85,B 0,C 180,E1 34921.376,E2 34921.376} C_VEL
LIN {X 0,Y 32.833,Z 1193.478,A -85,B 0,C 180,E1 34943.037,E2 34943.037} C_VEL
LIN {X 0,Y 17.127,Z 1194.454,A -85,B 0,C 180,E1 35010.025,E2 35010.025} C_VEL
LIN {X 0,Y 32.857,Z 1193.456,A -85,B 0,C 180,E1 35076.933,E2 35076.933} C_VEL
LIN {X 0,Y 75.589,Z 1188.441,A -85,B 0,C 180,E1 35098.505,E2 35098.505} C_VEL
LIN {X 0,Y 71.92,Z 1189.09,A -85,B 0,C 180,E1 35100.07,E2 35100.07} C_VEL
LIN {X 0,Y 32.366,Z 1194.258,A -85,B 0,C 180,E1 35120.934,E2 35120.934} C_VEL
LIN {X 0,Y 16.938,Z 1195.572,A -85,B 0,C 180,E1 35189.975,E2 35189.975} C_VEL
LIN {X 0,Y 23.296,Z 1194.961,A -85,B 0,C 180,E1 35243.046,E2 35243.046} C_VEL
LIN {X 0,Y 29.618,Z 1194.267,A -85,B 0,C 180,E1 35264.724,E2 35264.724} C_VEL
LIN {X 0,Y 38.492,Z 1193.3,A -85,B 0,C 180,E1 35277.928,E2 35277.928} C_VEL
LIN {X 0,Y 45.327,Z 1192.65,A -85,B 0,C 180,E1 35280.451,E2 35280.451} C_VEL
LIN {X 0,Y 45.352,Z 1192.612,A -85,B 0,C 180,E1 35281.934,E2 35281.934} C_VEL
LIN {X 0,Y 16.837,Z 1194.44,A -85,B 0,C 180,E1 35306.225,E2 35306.225} C_VEL
LIN {X 0,Y 9.184,Z 1194.714,A -85,B 0,C 180,E1 35370.047,E2 35370.047} C_VEL
LIN {X 0,Y 30.61,Z 1193.72,A -85,B 0,C 180,E1 35450.954,E2 35450.954} C_VEL
LIN {X 0,Y 45.369,Z 1192.575,A -85,B 0,C 180,E1 35457.98,E2 35457.98} C_VEL
LIN {X 0,Y 45.342,Z 1192.615,A -85,B 0,C 180,E1 35459.534,E2 35459.534} C_VEL
LIN {X 0,Y 16.524,Z 1194.896,A -85,B 0,C 180,E1 35483.798,E2 35483.798} C_VEL
LIN {X 0,Y 8.974,Z 1195.31,A -85,B 0,C 180,E1 35549.952,E2 35549.952} C_VEL
LIN {X 0,Y 38.492,Z 1193.3,A -85,B 0,C 180,E1 35637.928,E2 35637.928} C_VEL
LIN {X 0,Y 31.492,Z 1193.797,A -85,B 0,C 180,E1 35642.539,E2 35642.539} C_VEL
LIN {X 0,Y 2.839,Z 1194.927,A -85,B 0,C 180,E1 35667.854,E2 35667.854} C_VEL
LIN {X 0,Y 5.583,Z 1194.894,A -85,B 0,C 180,E1 35819.984,E2 35819.984} C_VEL
LIN {X 0,Y 0.987,Z 1195.048,A -85,B 0,C 180,E1 35909.563,E2 35909.563} C_VEL
LIN {X 0,Y 5.987,Z 1194.894,A -85,B 0,C 180,E1 35999.161,E2 35999.161} C_VEL
LIN {X 0,Y 1.237,Z 1194.975,A -85,B 0,C 180,E1 36090.349,E2 36090.349} C_VEL
LIN {X 0,Y 5.583,Z 1194.894,A -85,B 0,C 180,E1 36179.984,E2 36179.984} C_VEL
LIN {X 0,Y 7.576,Z 1196.893,A -85,B 0,C 180,E1 36183.309,E2 36183.309} C_VEL
LIN {X 0,Y 7.576,Z 1215,A -85,B 0,C 180,E1 36183.309,E2 36183.309} C_VEL
LIN {X 0,Y 7.576,Z 1215,A -85,B 0,C 180,E1 36183.309,E2 36183.309}

